% RSLogix 500 project I2A-JOB13A--MITCH_BAK059.RSS, saved by version 10.00.00.00 %
PROJECT "ML01B"    % processor: Bul.1763 MicroLogix 1100 Series B %

PROGRAM FILES
  LAD 2   9 rungs

DATA FILES
  O0 OUTPUT  4 elements
  I1 INPUT  6 elements
  S2 STATUS  66 elements
  B3 BINARY  1 elements
  T4 TIMER  1 elements
  C5 COUNTER  1 elements
  R6 CONTROL  1 elements
  N7 INTEGER  1 elements
  F8 FLOAT  1 elements

LADDER 2
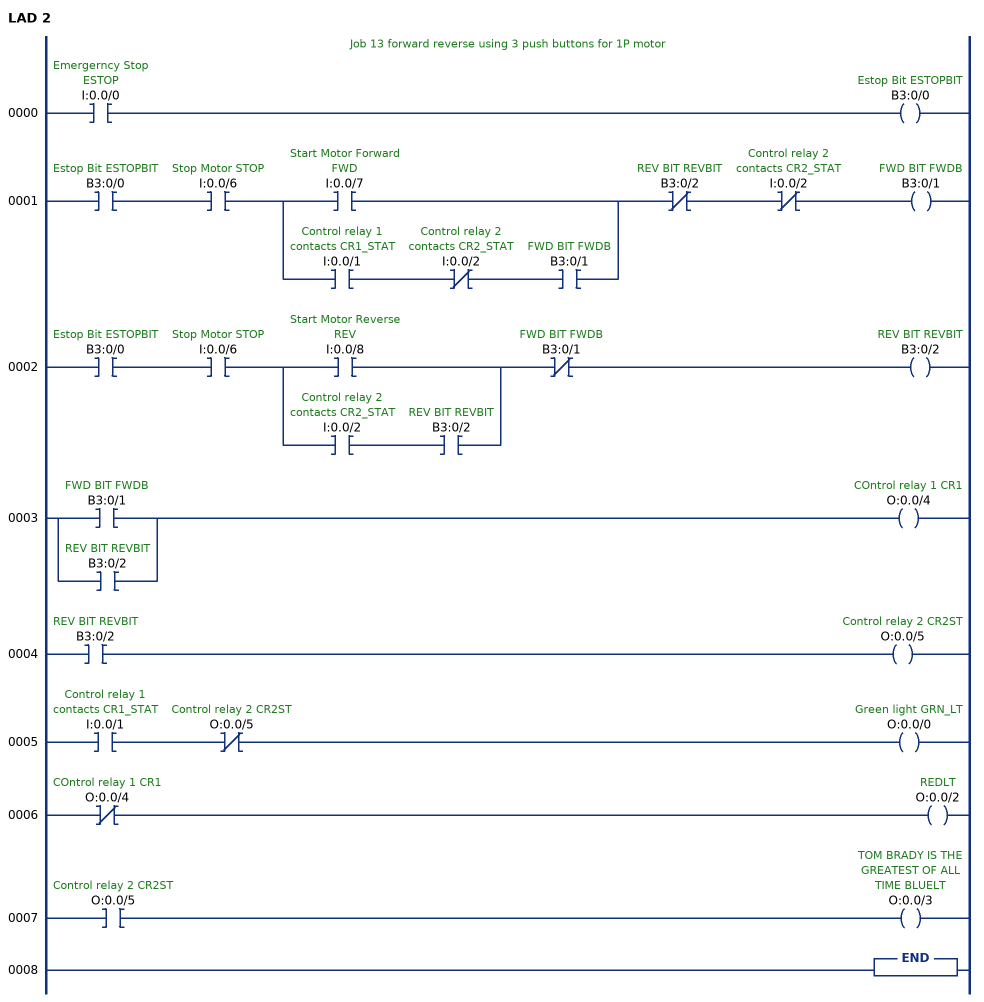
% Rung: 0 %
% Job 13 forward reverse using 3 push buttons for 1P motor %
SOR XIC I:0.0/0 OTE B3:0/0 EOR
%   I:0.0/0  ESTOP  "Emergerncy Stop" %
%   B3:0/0  ESTOPBIT  "Estop Bit" %
% Rung: 1 %
SOR XIC B3:0/0 XIC I:0.0/6 BST XIC I:0.0/7 NXB XIC I:0.0/1 XIO I:0.0/2 XIC B3:0/1 BND XIO B3:0/2 XIO I:0.0/2 OTE B3:0/1 EOR
%   B3:0/0  ESTOPBIT  "Estop Bit" %
%   I:0.0/6  STOP  "Stop Motor" %
%   I:0.0/7  FWD  "Start Motor Forward" %
%   I:0.0/1  CR1_STAT  "Control relay 1 contacts" %
%   I:0.0/2  CR2_STAT  "Control relay 2 contacts" %
%   B3:0/1  FWDB  "FWD BIT" %
%   B3:0/2  REVBIT  "REV BIT" %
% Rung: 2 %
SOR XIC B3:0/0 XIC I:0.0/6 BST XIC I:0.0/8 NXB XIC I:0.0/2 XIC B3:0/2 BND XIO B3:0/1 OTE B3:0/2 EOR
%   B3:0/0  ESTOPBIT  "Estop Bit" %
%   I:0.0/6  STOP  "Stop Motor" %
%   I:0.0/8  REV  "Start Motor Reverse" %
%   I:0.0/2  CR2_STAT  "Control relay 2 contacts" %
%   B3:0/2  REVBIT  "REV BIT" %
%   B3:0/1  FWDB  "FWD BIT" %
% Rung: 3 %
SOR BST XIC B3:0/1 NXB XIC B3:0/2 BND OTE O:0.0/4 EOR
%   B3:0/1  FWDB  "FWD BIT" %
%   B3:0/2  REVBIT  "REV BIT" %
%   O:0.0/4  CR1  "COntrol relay 1" %
% Rung: 4 %
SOR XIC B3:0/2 OTE O:0.0/5 EOR
%   B3:0/2  REVBIT  "REV BIT" %
%   O:0.0/5  CR2ST  "Control relay 2" %
% Rung: 5 %
SOR XIC I:0.0/1 XIO O:0.0/5 OTE O:0.0/0 EOR
%   I:0.0/1  CR1_STAT  "Control relay 1 contacts" %
%   O:0.0/5  CR2ST  "Control relay 2" %
%   O:0.0/0  GRN_LT  "Green light" %
% Rung: 6 %
SOR XIO O:0.0/4 OTE O:0.0/2 EOR
%   O:0.0/4  CR1  "COntrol relay 1" %
%   O:0.0/2  REDLT %
% Rung: 7 %
SOR XIC O:0.0/5 OTE O:0.0/3 EOR
%   O:0.0/5  CR2ST  "Control relay 2" %
%   O:0.0/3  BLUELT  "TOM BRADY IS THE GREATEST OF ALL TIME" %
% Rung: 8 %
SOR END EOR

OTHER DOCUMENTED ADDRESSES
  I:0.0/3  DIRECTION  "Direction Forward- off-Reverse"
  I:0.0/4  3PSS_B  "Three posision selector switch B"
  I:0.0/5  2PSSA  "2 position selector switch A"
  O:0.0/1  YELLOWLT

DATA TABLE (non-zero values as saved)
DATA B3
% B3:0 % 0X0001
DATA T4
% .PRE .ACC %
% T4:0 % 8 0
